ABB RobotStudio station: practica5_EstacionDePartida.rspag

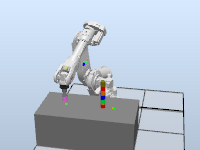
--- station ---
Station practica3_EstacionDePartida (saved by RobotStudio 20.4.9280.0)
Controller Sistema6
  mechanical unit ROB_1: IRB6640_180_255__04, 6 joints, base frame (0, 0, 0) mm
Layout (positions relative to the parent item):
  - Ventosa [mechanism] at (1500, -500, 1150) mm, rotated rx 180 ry 0 rz 180 deg
      TCP Ventosa at (0, 0, 200) mm
      links: PiezaVentosa
  - IRB6640_180_255__04 [mechanism, from Robots\IRB6640_180_255_G_04.rslib] at (0, 0, 0) mm; joint values [-0.3218, 0.1942, 0.4103, 0, 0.9663, -0.3218] (rad or m)
  - MesaTrabajoParteIzq [part]
  - MesaTrabajoParteDer [part]
  - CI_VentosaVacuostato [smart component]
      signals: DI ActivaVentosa, DO Vacuostato
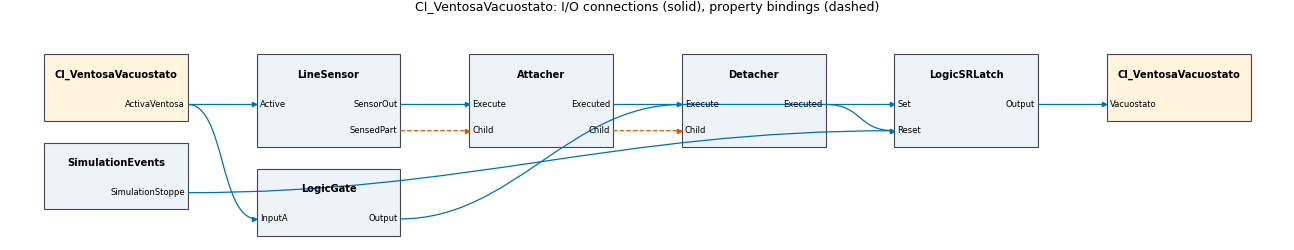
      connections:
        CI_VentosaVacuostato.ActivaVentosa -> LineSensor.Active
        LineSensor.SensorOut -> Attacher.Execute
        Attacher.Executed -> LogicSRLatch.Set
        LogicSRLatch.Output -> CI_VentosaVacuostato.Vacuostato
        Detacher.Executed -> LogicSRLatch.Reset
        SimulationEvents.SimulationStopped -> LogicSRLatch.Reset
        CI_VentosaVacuostato.ActivaVentosa -> LogicGate.InputA
        LogicGate.Output -> Detacher.Execute
        LineSensor.SensedPart => Attacher.Child
        Attacher.Child => Detacher.Child
    - LineSensor [smart component, from Components\LineSensor.rslib] at (1500, -500, 950) mm, rotated rx 180 ry 0 rz 180 deg
        properties: Start=[0 0 -0.002]; End=[0 0 0.02]; Radius=0.002; SensedPart=MesaTrabajoParteDer; SensedPoint=[1.5 -0.5 0.75]
      - _sensorPart_ [part]
    - SimulationEvents [smart component, from Components\SimulationEvents.rslib]
    - LogicSRLatch [smart component, from Components\LogicSRLatch.rslib]
    - Attacher [smart component, from Components\Attacher.rslib]
        properties: Parent=Ventosa; Flange=0; Child=MesaTrabajoParteDer; Mount=false; Offset=[0 0 0]; Orientation=[0 0 0]
    - Detacher [smart component, from Components\Detacher.rslib]
        properties: Child=MesaTrabajoParteDer; KeepPosition=true
    - LogicGate [smart component, from Components\LogicGate.rslib]
        properties: Operator=NOT; Delay=0.1
  - Pieza_8 [part] at (0, -1000, 98.56) mm
  - Pieza_15 [part] at (0, -200, 407.51) mm
  - Pieza_16 [part] at (0, -200, 209.94) mm
  - Pieza_17 [part] at (0, -200, 12.99) mm
  - Pieza_18 [part] at (0, -200, -192.07) mm
  - Pieza_19 [part] at (0, -200, -391.25) mm
  - Pieza_20 [part] at (0, -200, -584.44) mm
Attachment: LineSensor is attached to Ventosa / PiezaVentosa
Attachment: Ventosa is attached to IRB6640_180_255__04 / Link6
Attachment: Pieza_8 is attached to Ventosa / PiezaVentosa
Station logic (signal -> signal, property => property):
  CI_VentosaVacuostato.Vacuostato -> Sistema6.ED_PiezaCogida
  Sistema6.SD_ActivaVentosa -> CI_VentosaVacuostato.ActivaVentosa

--- Backups/Sistema6/RAPID/TASK1/PROGMOD/CalibData.mod ---
MODULE CalibData
	PERS tooldata Ventosa:=[TRUE,[[0,0,200],[1,0,0,0]],[1,[0,0,125],[1,0,0,0],0.002,0.002,0.0013]];
ENDMODULE

--- Backups/Sistema6/RAPID/TASK1/PROGMOD/Module1.mod ---
MODULE Module1
	CONST robtarget pReposo:=[[1808.910161514,0,1855],[0.5,0,0.866025404,0],[0,0,0,0],[9E+09,9E+09,9E+09,9E+09,9E+09,9E+09]];
	CONST robtarget pBaseTorre1:=[[1500,500,750],[0,0,1,0],[0,0,0,0],[9E+09,9E+09,9E+09,9E+09,9E+09,9E+09]];
    CONST robtarget pBaseTorre2:=[[1500,-500,750],[0,0,1,0],[0,0,0,0],[9E+09,9E+09,9E+09,9E+09,9E+09,9E+09]];

    CONST num diametro := 100;
    CONST num altura := 100;



PROC main()
    ! Movemos la primera torre de 7 piezas 2 veces el diametro de la pieza
    MueveTorre pBaseTorre1, pBaseTorre2, 7, -2;

ENDPROC

PROC MueveTorre(robtarget pOrigen,robtarget pDestino, num nPiezas, num desplazamiento)
    VAR num AlturaEnOrigen := 0;
    VAR num AlturaEnDestino := 0;
    VAR num nPiezas2 := 0;
    VAR robtarget pApoyo;
    VAR robtarget pInter;
    VAR robtarget pAproxOrigen;
    VAR robtarget pAproxDestino;
    VAR robtarget pOrigen2;

    !Calculamos la altura en el origen y en destino
    AlturaEnOrigen := nPiezas * altura;
    AlturaEnDestino := AlturaEnDestino + altura;
    nPiezas2 := nPiezas;

    !Calculamos los puntos de aproximacion
    pAproxOrigen := Offs (pOrigen, 0, 0, AlturaEnOrigen + altura); !Hacemos el punto
    pAproxDestino := Offs (pOrigen, 0, desplazamiento * diametro, AlturaEnOrigen + altura); !Hacemos el punto

    !Bucle while
    WHILE nPiezas2 > 0 DO

    !Movemos el brazo a la posición de aproximacion
    MoveL pAproxOrigen,v1000,z0,Ventosa\WObj:=wobj0;

    !Movemos la ventosa a la primera pieza
    pApoyo := Offs (pOrigen, 0, 0, AlturaEnOrigen); !Hacemos el punto
    MoveLDO pApoyo,v2000,fine,Ventosa\WObj:=wobj0,SD_ActivaVentosa,1;
    WaitDI ED_PiezaCogida, 1; !Esperamos a que PiezaCogida esté a 1, así no esperamos los dos segundos
    MoveL pAproxOrigen,v2000,z0,Ventosa\WObj:=wobj0;

    !Movemos a la posición de aproximacion
    MoveL pAproxDestino,v2000,z0,Ventosa\WObj:=wobj0;

    !Movemos a donde queramos moverlo
    pInter := Offs (pOrigen, 0, desplazamiento * diametro, AlturaEnDestino); !Hacemos el punto
    MoveLDO pInter,v2000,fine,Ventosa\WObj:=wobj0,SD_ActivaVentosa,0;
    MoveL pAproxDestino,v2000,z0,Ventosa\WObj:=wobj0;

    !Calculamos la altura del origen y del destino
    nPiezas2 := nPiezas2 - 1;
    AlturaEnOrigen := nPiezas2 * altura;
    AlturaEnDestino := AlturaEnDestino + altura;

    ENDWHILE

    !Volvemos a resetear el numero de piezas
    nPiezas2 := nPiezas;
    AlturaEnOrigen := nPiezas2 * altura;
    AlturaEnDestino := 0 + altura;

    !Ponemos como punto origen el nuevo punto
    pOrigen2 := Offs (pOrigen, 0, desplazamiento * diametro, AlturaEnDestino + altura);

    !Calculamos los puntos de aproximacion
    pAproxOrigen := Offs (pOrigen2, 0, 0, altura * nPiezas2); !Hacemos el punto
    pAproxDestino := Offs (pDestino, 0, 0, AlturaEnDestino + altura); !Hacemos el punto

    !Volvemos a rehacer el bucle while
    WHILE nPiezas2 > 0 DO

    !Movemos el brazo a la posición de aproximacion
    MoveL pAproxOrigen,v2000,z0,Ventosa\WObj:=wobj0;

    !Movemos la ventosa a la primera pieza
    pApoyo := Offs (pOrigen2, 0, 0, AlturaEnOrigen - (altura * 2)); !Hacemos el punto
    MoveLDO pApoyo,v2000,fine,Ventosa\WObj:=wobj0,SD_ActivaVentosa,1;
    WaitDI ED_PiezaCogida, 1; !Esperamos a que PiezaCogida esté a 1, así no esperamos los dos segundos
    MoveL pAproxOrigen,v2000,z0,Ventosa\WObj:=wobj0;

    !Movemos a la posición de aproximacion
    MoveL pAproxDestino,v2000,z0,Ventosa\WObj:=wobj0;

    !Movemos a donde queramos moverlo
    MoveLDO pDestino,v2000,fine,Ventosa\WObj:=wobj0,SD_ActivaVentosa,0;
    MoveL pAproxDestino,v500,z0,Ventosa\WObj:=wobj0;

    !Calculamos la altura del origen y del destino
    nPiezas2 := nPiezas2 - 1;
    AlturaEnOrigen := nPiezas2 * altura;
    AlturaEnDestino := AlturaEnDestino + altura;

    ENDWHILE




ENDPROC

ENDMODULE

--- Backups/Sistema6/RAPID/TASK1/SYSMOD/LINKEDM.sys ---
%%%
  VERSION:1
  LANGUAGE:ENGLISH
%%%

MODULE LINKEDM (SYSMODULE)

! FOLLOWER
!     Name of electronically linked follower axis used by operator at teach pendent.
      PERS string l_f_axis_name{5}       :=  ["",  "", "", "", ""];

!     Name of the mechanical unit for follower axis.
      PERS string l_f_mecunt_n{5}  :=  ["", "", "", "", ""];

!     Linked follower axis number in the mechanical unit (first axis in mech. unit is number 1).
      PERS num l_f_axis_no{5}      :=  [0,          0,   0,  0,  0];

! MASTER
!     Name of the mechanical unit for linked master axis.
      PERS string l_m_mecunt_n{5} :=  ["", "", "", "", ""];

!     Linked master axis number in the mechanical unit (first axis in mech. unit is number 1).
!     See axis number table in documentation for different master mechanical units.
      PERS num l_m_axis_no{5}     :=  [0,  0,  0,  0,  0];

! POSITION OFFSET
!     The increase of the allowed offset position between the master and follower
!     positions, used when starting AUTO mode. As soon as the offset is decreased
!     the old configurated parameter is used.
!     Example: 3 => the configurated value of allowed offset is increased 3 times.
      PERS num offset_ratio{5}       :=  [10,  10,   10,  10,  10];

! SPEED RATIO
!     Speed_ratio used in AUTO and JOG modes [ very_slow   slow    normal    fast]
!     Value 1 = max allowed manual speed.
      CONST num speed_ratio {20}      := [0.01, 0.01, 0.01, 0.01, 0.01,
                                          0.05, 0.05, 0.05, 0.05, 0.05,
                                          0.20, 0.20, 0.20, 0.20, 0.20,
                                          1.00, 1.00, 1.00, 1.00, 1.00];

! STEP SIZE
!     Displacement position used in JOG mode for each activation of positive or
!     negative movement.                  [very_short    short   normal   long]
!     Unit degees or meter.
      CONST num displacement {20}     := [0.001, 0.001, 0.001, 0.001, 0.001,
                                          0.005, 0.005, 0.005, 0.005, 0.005,
                                          0.020, 0.020, 0.020, 0.020, 0.020,
                                          0.100, 0.100, 0.100, 0.100, 0.100];


!-------------------------------------------------------------
 PROC Linked_m ()
      Linked_m_exe ;
 ENDPROC
ENDMODULE

--- Backups/Sistema6/SYSPAR/EIO.cfg ---
EIO:CFG_1.0:6:1::
#
INDUSTRIAL_NETWORK:

      -Name "DeviceNet" -Label "DeviceNet Master/Slave Network" -Address "2"
#
DEVICENET_DEVICE:

      -Name "MiDeviceNet" -Label "MiDeviceNet"
#
DEVICENET_INTERNAL_DEVICE:

      -Name "DN_Internal_Device" -VendorName "ABB Robotics"\
      -ProductName "DeviceNet Internal Slave Device"
#
EIO_SIGNAL:

      -Name "ED_PiezaCogida" -SignalType "DI" -Device "MiDeviceNet"\
      -Label "ED_PiezaCogida" -DeviceMap "0" -Access "All"

      -Name "SD_ActivaVentosa" -SignalType "DO" -Device "MiDeviceNet"\
      -Label "SD_ActivaVentosa" -DeviceMap "0" -Access "All"
